// TIA Portal project "Semaforo V2" (V17)

(* hardware
DEVICE "S7-400 station_1"  S7-400 station
   slot 0: "UR1_0"  UR1  6ES7 400-1TA01-0AA0
   slot 1: "PS 407 4A_1"  PS 407 4A  6ES7 407-0DA02-0AA0
   slot 2: "PLC_1"  CPU 416-3 PN/DP  6ES7 416-3ES07-0AB0  V7.0
      slot 2: "MPI/DP interface_1"  X1
      slot 5: "PROFINET interface_1"  PN-IO
         slot 1: "Port_1"  Port
         slot 2: "Port_2"  Port
*)

// ===== PLC "PLC_1"  CPU 416-3 PN/DP =====

VAR_GLOBAL   // PLC tag table "Default tag table"
   "Tag_1" AT %I0.0 : Bool;
   "Tag_2" AT %Q0.0 : Bool;
   "Tag_3" AT %Q0.1 : Bool;
   "Tag_4" AT %Q0.2 : Bool;
   "Tag_5" AT %Q0.6 : Bool;
   "Tag_6" AT %Q0.5 : Bool;
   "Tag_7" AT %Q0.4 : Bool;
   "Tag_8" AT %Q0.3 : Bool;
   "Tag_9" AT %Q0.7 : Bool;
   "Tag_10" AT %M0.0 : Bool;
   "Tag_11" AT %M0.1 : Bool;
   "Tag_12" AT %I0.1 : Bool;
   "Tag_13" AT %M0.2 : Bool;
   "Tag_14" AT %M0.4 : Bool;
   "Pisca" AT %M1.5 : Bool;
   "Tag_15" AT %M0.5 : Bool;
   "Tag_16" AT %I0.2 : Bool;
END_VAR

DATA_BLOCK "Block_STL_DB"   // DB1
{ S7_Optimized_Access := 'FALSE' }
VERSION : 0.1
// stored: InstanceOfName Block_STL
"Block_STL"
BEGIN
END_DATA_BLOCK

FUNCTION_BLOCK "Block_STL"   // FB1, STL
{ S7_Optimized_Access := 'FALSE' }
VERSION : 0.1
   VAR_INPUT
      Liga_Desliga : Bool;
      Botao_Pedestre : Bool;
   END_VAR
   VAR_OUTPUT
      A_Vermelho : Bool;
      A_Amarelo : Bool;
      A_Verde : Bool;
      B_Vermelho : Bool;
      B_Amarelo : Bool;
      B_Verde : Bool;
      P_Vermelho : Bool;
      P_Verde : Bool;
   END_VAR
   VAR
      Auxiliar_Pedestre1 : Bool;
      Auxiliar_Pedestre2 : Bool;
   END_VAR
BEGIN

REGION Network 1: Start
   //Loop

         A     #Liga_Desliga;
         A(;
         AN    "TON5".Q;
         O     #Auxiliar_Pedestre2;
         );
         AN    "TONP2".Q;
         =     "TON2".IN;

         S     #A_Verde;
         S     #B_Vermelho;
         S     #P_Vermelho;
END_REGION

REGION Network 2: Primeiro ciclo: Semáforo A
         CALL  TON , "TON2"
         ( IN := ,
           PT := T#5S,
           Q  := ,
           ET :=
         );

         A     "TON2".Q;
         R     #A_Verde;
         S     #A_Amarelo;

         CALL  TON , "TON3"
         ( IN := "TON2".Q,
           PT := T#2S,
           Q  := ,
           ET :=
         );

         A     "TON3".Q;
         R     #A_Amarelo;
         S     #A_Vermelho;
END_REGION

REGION Network 3: Verificação de Pedestre
         A     #Botao_Pedestre;
         AN    "TON3".Q;
         S     #Auxiliar_Pedestre1;

         A     #Auxiliar_Pedestre1;
         A     "TON3".Q;
         =     "TONP1".IN;
         R     #P_Vermelho;
         S     #P_Verde;

         CALL  TON , "TONP1"
         ( IN := ,
           PT := T#7S,
           Q  := ,
           ET :=
         );

         A     "TONP1".Q;
         R     #P_Verde;
         S     #P_Vermelho;
         R     #Auxiliar_Pedestre1;
END_REGION

REGION Network 4: Segundo ciclo: Semáforo B
   //Inicio do segundo ciclo
         A     "TON3".Q;
         AN    #Auxiliar_Pedestre1;
         =     "TON4".IN;
         R     #B_Vermelho;
         R     #P_Verde;
         S     #B_Verde;

         CALL  TON , "TON4"
         ( IN := ,
           PT := T#5S,
           Q  := ,
           ET :=
         );

         A     "TON4".Q;
         R     #B_Verde;
         S     #B_Amarelo;

         CALL  TON , "TON5"
         ( IN := "TON4".Q,
           PT := T#2S,
           Q  := ,
           ET :=
         );

         A     "TON5".Q;
         R     #B_Amarelo;
         S     #B_Vermelho;
END_REGION

REGION Network 5: Verificação de Pedestre
   //Fim do segundo ciclo: Pedestre 2
         A     #Botao_Pedestre;
         A     "TON3".Q;
         S     #Auxiliar_Pedestre2;

         A     #Auxiliar_Pedestre2;
         A     "TON5".Q;
         =     "TONP2".IN;
         R     #P_Vermelho;
         S     #P_Verde;

         CALL  TON , "TONP2"
         ( IN := ,
           PT := T#7S,
           Q  := ,
           ET :=
         );
         A     "TONP2".Q;
         R     #P_Verde;
         S     #P_Vermelho;
         R     #Auxiliar_Pedestre2;
END_REGION

REGION Network 6
         AN    #Auxiliar_Pedestre2;
         A     "TON5".Q;
         R     #A_Vermelho;
         R     #B_Vermelho;
END_REGION
END_FUNCTION_BLOCK

ORGANIZATION_BLOCK "Main"   // OB1, LAD
TITLE = "Main Program Sweep (Cycle)"
{ S7_Optimized_Access := 'FALSE' }
VERSION : 0.1
   VAR_TEMP
      OB1_EV_CLASS : Byte;   // Bits 0-3 = 1 (Coming event), Bits 4-7 = 1 (Event class 1)
      OB1_SCAN_1 : Byte;   // 1 (Cold restart scan 1 of OB 1), 3 (Scan 2-n of OB 1)
      OB1_PRIORITY : Byte;   // Priority of OB Execution
      OB1_OB_NUMBR : Byte;   // 1 (Organization block 1, OB1)
      OB1_RESERVED_1 : Byte;   // Reserved for system
      OB1_RESERVED_2 : Byte;   // Reserved for system
      OB1_PREV_CYCLE : Int;   // Cycle time of previous OB1 scan (milliseconds)
      OB1_MIN_CYCLE : Int;   // Minimum cycle time of OB1 (milliseconds)
      OB1_MAX_CYCLE : Int;   // Maximum cycle time of OB1 (milliseconds)
      OB1_DATE_TIME : Date_And_Time;   // Date and time OB1 started
   END_VAR
BEGIN

REGION Network 1
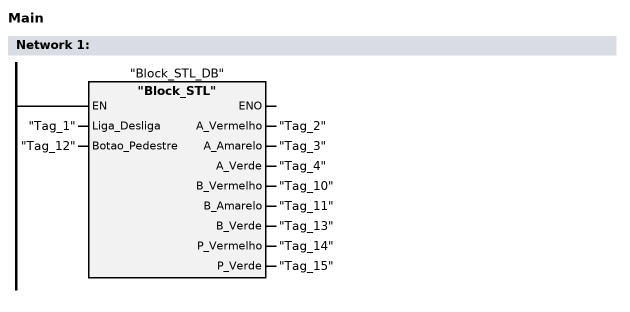
   RUNG wire#powerrail
      "Block_STL_DB"(Liga_Desliga := "Tag_1", Botao_Pedestre := "Tag_12", A_Vermelho => "Tag_2", A_Amarelo => "Tag_3", A_Verde => "Tag_4", B_Vermelho => "Tag_10", B_Amarelo => "Tag_11", B_Verde => "Tag_13", P_Vermelho => "Tag_14", P_Verde => "Tag_15")
   END_RUNG
   // the same network as SCL:
   "Block_STL_DB"(Liga_Desliga := "Tag_1",   // "Block_STL"
                  Botao_Pedestre := "Tag_12",
                  A_Vermelho => "Tag_2",
                  A_Amarelo => "Tag_3",
                  A_Verde => "Tag_4",
                  B_Vermelho => "Tag_10",
                  B_Amarelo => "Tag_11",
                  B_Verde => "Tag_13",
                  P_Vermelho => "Tag_14",
                  P_Verde => "Tag_15");
END_REGION
END_ORGANIZATION_BLOCK